// TIA Portal V16 export
// export: Created 2026-03-31T12:42:57.2749443Z, ExportSetting WithDefaults, DisplayName Totally Integrated Automation Portal, DisplayVersion V16, DisplayName TIA Portal Version Control Interface, DisplayVersion V16, DisplayName TIA Portal Openness, DisplayVersion V16, DisplayName STEP 7 Professional, DisplayVersion V16, DisplayName STEP 7 Safety, DisplayVersion V16, DisplayName WinCC Advanced, DisplayVersion V16
ORGANIZATION_BLOCK "OB80"   // OB80, FBD, TimeErrorInterrupt
VERSION : 0.1
// stored: IsIECCheckEnabled false
   VAR_TEMP
      Temp_0 : Byte;
      Temp_1 : Byte;
      Temp_2 : Byte;
      Temp_3 : Byte;
      Temp_4 : Byte;
      Temp_5 : Byte;
      Temp_6 : Word;
      Temp_7 : Byte;
      Temp_8 : Byte;
      Temp_9 : Byte;
      Temp_10 : Byte;
      Temp_11 : Date_And_Time;
   END_VAR
BEGIN
END_ORGANIZATION_BLOCK
